// TwinCAT 3 PLC project MAS418_PLC
// ProgramVersion: 3.1.4024.0
// libraries:
//   Tc2_Standard, * (Beckhoff Automation GmbH)
//   Tc2_System, * (Beckhoff Automation GmbH)
//   Tc3_Module, * (Beckhoff Automation GmbH)
// project tree:
//   / GlobalTextList.TcGTLO, PlcTask.TcTTO, Visualization Manager.TcVMO (not stored)
//   POUs/ MAIN.TcPOU
//   VISUs/ HMI.TcVIS
// real-time tasks:
//   TASK PlcTask: cycle T#10ms, priority 20, ADS port 350

CONFIGURATION MAS418_PLC
    RESOURCE PLC ON TwinCAT3
        TASK PlcTask(INTERVAL := T#10ms, PRIORITY := 20);
        PROGRAM MAIN WITH PlcTask : MAIN;
    END_RESOURCE
END_CONFIGURATION

// ---- POUs/MAIN.TcPOU
PROGRAM MAIN
VAR
	bEnable : BOOL;
	bStart : BOOL;
	nINT : INT := -32768;
	nUINT : UINT := 65535;
	fREAL : REAL := 255.255;
END_VAR

bEnable := bStart;

END_PROGRAM

// ---- GlobalTextList.TcGTLO
TEXTLIST GlobalTextList
  152 = 'BOOL'
  794 = 'BOOL:%s'
  177 = 'DataTypeTesting'
  898 = 'INT'
  20 = 'Power ON'
  849 = 'REAL'
  104 = 'STRING'
  30 = 'UINT'
END_TEXTLIST

// ---- VISUs/HMI.TcVIS
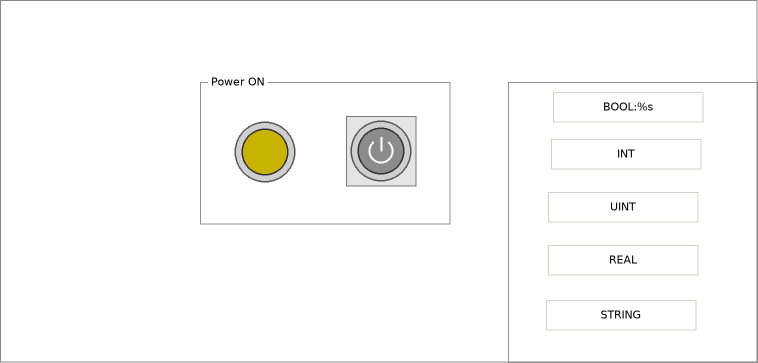
VISUALIZATION HMI  // 758x363
    GroupBox (200,74 250x150), "Power ON"
        Lamp1 (30,43 70x70), variable: MAIN.bEnable, style: Lamp-Lamp1-Yellow
        PowerSwitch (146,42 70x70), variable: MAIN.bStart, behaviour: TOGGLE, style: Switch-PowerSwitch-Gray
    GroupBox (508,74 250x289)
        Textfield (45,18 150x30), "BOOL:%s", text variable: MAIN.bEnable
        Textfield (43,65 150x30), "INT"
        Textfield (40,118 150x30), "UINT"
        Textfield (40,171 150x30), "REAL"
        Textfield (38,226 150x30), "STRING"
END_VISUALIZATION
